FUNCTION_BLOCK FB_EtherCATReader
VAR_INPUT
		ID : USINT;
END_VAR
VAR_OUTPUT
	WrittenAll : BOOL := FALSE;
END_VAR

VAR
	SymInfo  : PLC_ReadSymInfo;
	VarSymInfo  :  PLC_ReadSymInfoByName;
	Exec : BOOL;
	
	DataInt : DINT;
	//RecievedData : ARRAY [1..256] OF INT; //used to count reads of each parameter
	i : INT;
	ParametersWritten : USINT;
	RefreshParameters : BOOL := FALSE;
	
	ParameterID_FromMom AT %I* : USINT;
	ParameterWord_FromMom AT %I* : DINT; //ParameterWord cycles through many arrays to send less time critical data
	ParameterID_ToMom AT %Q* : USINT;
END_VAR

//ParameterWord_FromMom consists of 32 bytes. The first(greatest) 8 bytes ID the Variable to write and the last 24 include the data. 
// ParameterID		Parameter To Write					Format
// 1				GVL_Motion.lrEncoder_ScalingNum		1/DATAINT := ScalingNum
// 2				GVL_Index.Admin_Max					:= 512 * DataInt (largest bit is sign)	
// 3				GVL_Index.Admin_Min					:= 	512 * DataInt (largest bit is sign)	
// 4				GVL_Index.Direction_Flipped			>0 		
// 5				GVL_Motion.lrDistance_1_Motor_Rev	:= ?????????????????????????
// 6				GVL_Speeds.QuickStop_Accel		
// 7 				GVL_Speeds.lrDecel_For_EStop		:=?
SymInfo(Port:=851, Start:=Exec);
VarSymInfo(Port:=851, SymName:= 'P30_MAIN.execute', Start:=Exec);

DataInt := Parameterword_FromMom ;
ID := ParameterID_FromMom ;

CASE ID OF
//1: 	GVL_Motion.lrEncoder_ScalingNum := 1/DINT_TO_LREAL(DataInt);
2: 	GVL_Index.Home_Switch_Offset := DataInt ;
3: 	GVL_Index.Admin_Min :=  DataInt ;
4:  GVL_Index.Direction_Flipped := DataInt > 0;
5: 	GVL_Motion.lrDistance_1_Motor_Rev := DataInt;
//6:	GVL_Speeds.QuickStop_Accel := DataInt;
//7:	GVL_Speeds.lrDecel_For_EStop := DataInt;
	
ELSE
	ID := 0;
END_CASE

ParameterID_ToMom := ParameterID_FromMom;

//RecievedData[ID] := RecievedData[ID] + 1;

ParametersWritten := 0;
FOR i := 1 TO 256 DO
//	IF RefreshParameters THEN RecievedData[i] := 0;  END_IF	
	//IF RecievedData[i] > 0 THEN ParametersWritten := ParametersWritten + 1; END_IF
END_FOR

IF RefreshParameters THEN RefreshParameters := FALSE; END_IF

END_FUNCTION_BLOCK

(* stored: Version 1.1.0.1, ProductVersion 3.1.4022.3
   POU FB_EtherCATReader: Id {1d3ebd30-390d-4f3c-93df-f8f5b484e808}, SpecialFunc None *)
